// TIA Portal V18 export
FUNCTION_BLOCK "Utility_PID"   // FB2, FBD
TITLE = Utility PID Control
{ S7_Optimized_Access := 'TRUE' }
VERSION : 0.1
// Utility PID Control
// stored: AutoNumber true, IsIECCheckEnabled false, IsRetainMemResEnabled false, MemoryReserve 100, SetENOAutomatically false, UDAEnableTagReadback false
   VAR_INPUT
      START : Bool;
      SP : Real;
      PV : Real;
      CONTROL_MODE : Int;
      "TIME" : Int;
      PRE_SP : Int;
      AM : Bool;
      P : Int;
      I : Int;
      D : Int;
      JAC_IN : Real;
      JAC_OUT : Real;
      HHSP : Real;
      HSP : Real;
      LSP : Real;
      LLSP : Real;
      PIDRST : Bool;
      SOURCE_SEL : Int;
      AIR_XV_OPN : Bool;
      BYP_XV_OPN : Bool;
      VENT_OPN : Bool;
      CONDENSATE_XV_OPN : Bool;
      DRAIN_XV_OPN : Bool;
      SCV_XV_OPN : Bool;
   END_VAR
   VAR_OUTPUT
      START_PV : Real;
      CVOUT : Int;
      SCVOUT : Real;
      STATUS : Int;
      RAMP_SP : Real;
      JSP : Real;
      PID_PV : Real;
      RUN_MIN : Int;
      RUN_HR : Int;
      STEAM_SCVOUT : Real;
      STEAM_CVOUT : Int;
   END_VAR
   VAR_IN_OUT
      PAUSE : Bool;
      MAN_OUT : Real;
      TEMP_LIMIT : Real;
      STEAM_MAN_OUT : Real;
   END_VAR
   VAR
      RAMP_MODE : Bool;
      MAINT_MODE : Bool;
      J_MAINT_MODE : Bool;
      NO_RAMP : Bool;
      HEAT_COOL : Bool;
      BSTBIT : Bool;
      HOLD : Int;
      RAMP : Real;
      RAMP_RST : Bool;
      RMPSTART : Bool;
      Ramp_Substitute : Real;
      RAMP_INIT_RST : Bool;
      JKT_RAMP : Bool;
      MASS_CONTROL : Bool;
      TIMER_TRIG : Bool;
      iSTEAM_SCVOUT : Real;
      iSTEAM_CVOUT : Int;
      iSTEAM_SCV_SCL : Real;
      iSTEAM_CV_SCL : Int;
      iDRAIN_UP : Bool;
   END_VAR
BEGIN

REGION Network 1: Mode Selection
   // Mode Selection
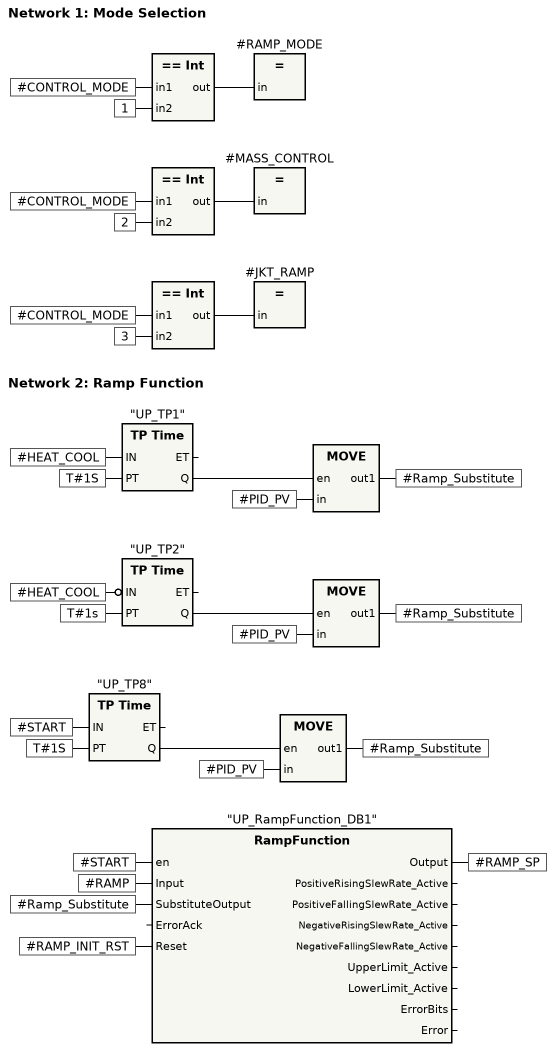
   #RAMP_MODE := #CONTROL_MODE = 1;
   #MASS_CONTROL := #CONTROL_MODE = 2;
   #JKT_RAMP := #CONTROL_MODE = 3;
END_REGION

REGION Network 2: Ramp Function
   // Ramp Function
   "UP_TP1".TP(IN := #HEAT_COOL, PT := T#1S);
   IF "UP_TP1".Q THEN #Ramp_Substitute := #PID_PV; END_IF;
   "UP_TP2".TP(IN := NOT #HEAT_COOL, PT := T#1s);
   IF "UP_TP2".Q THEN #Ramp_Substitute := #PID_PV; END_IF;
   "UP_TP8".TP(IN := #START, PT := T#1S);
   IF "UP_TP8".Q THEN #Ramp_Substitute := #PID_PV; END_IF;
   IF #START THEN
       "UP_RampFunction_DB1"(Input := #RAMP,   // RampFunction
                             SubstituteOutput := #Ramp_Substitute,
                             Reset := #RAMP_INIT_RST,
                             Output => #RAMP_SP);
   END_IF;
END_REGION

REGION Network 3: Ramp Reset
   // Ramp Reset
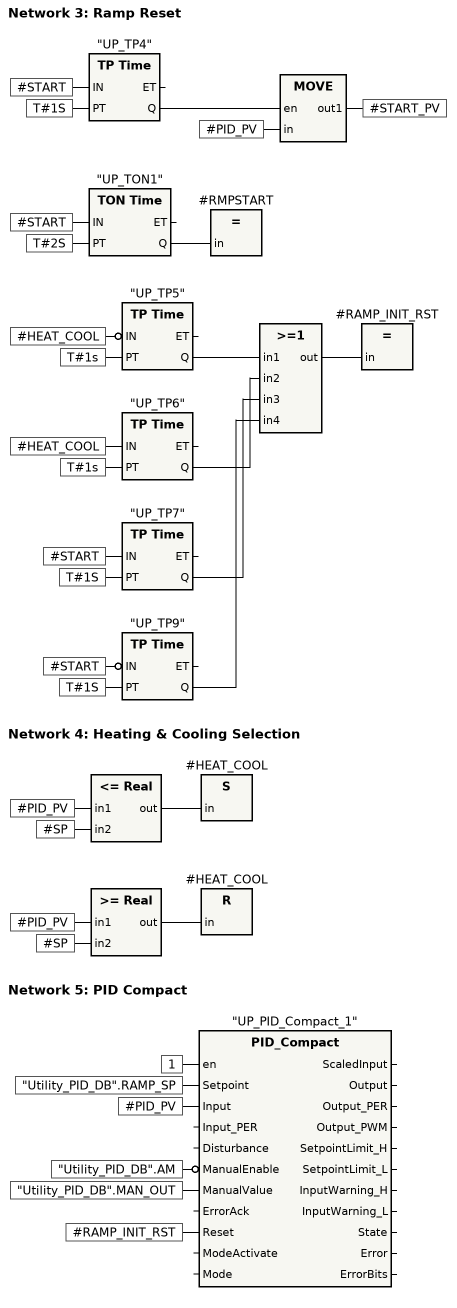
   "UP_TP4".TP(IN := #START, PT := T#1S);
   IF "UP_TP4".Q THEN #START_PV := #PID_PV; END_IF;
   "UP_TON1".TON(IN := #START, PT := T#2S);
   #RMPSTART := "UP_TON1".Q;
   "UP_TP5".TP(IN := NOT #HEAT_COOL, PT := T#1s);
   "UP_TP6".TP(IN := #HEAT_COOL, PT := T#1s);
   "UP_TP7".TP(IN := #START, PT := T#1S);
   "UP_TP9".TP(IN := NOT #START, PT := T#1S);
   #RAMP_INIT_RST := "UP_TP5".Q OR "UP_TP6".Q OR "UP_TP7".Q OR "UP_TP9".Q;
END_REGION

REGION Network 4: Heating & Cooling Selection
   // Heating & Cooling Selection
   IF #PID_PV <= #SP THEN #HEAT_COOL := TRUE; END_IF;
   IF #PID_PV >= #SP THEN #HEAT_COOL := FALSE; END_IF;
END_REGION

REGION Network 5: PID Compact
   IF 1 THEN
       "UP_PID_Compact_1"(Setpoint := "Utility_PID_DB".RAMP_SP,   // PID_Compact
                          Input := #PID_PV,
                          ManualEnable := NOT "Utility_PID_DB".AM,
                          ManualValue := "Utility_PID_DB".MAN_OUT,
                          Reset := #RAMP_INIT_RST);
   END_IF;
END_REGION

REGION Network 6 (SCL): Moving
   (* PID Parameters Moving *)
   "UP_PID_Compact_1".Retain.CtrlParams.Gain:= #P;
   "UP_PID_Compact_1".Retain.CtrlParams.Ti := #I;
   "UP_PID_Compact_1".Retain.CtrlParams.Td := #D;

   #RAMP := #SP;

   IF #RAMP_MODE OR #MASS_CONTROL THEN
       #PID_PV := #PV;
   END_IF;
   IF #JKT_RAMP THEN
       #PID_PV := #JAC_IN;
   END_IF;


   IF #AM = 1 AND #START = 1 AND #SOURCE_SEL<>5 THEN
       #SCVOUT := "UP_PID_Compact_1".Output;
       #CVOUT := "UP_PID_Compact_1".Output_PER;
   END_IF;
   IF (#AM = 1 AND #START = 0 ) OR (#AM = 1 AND #SOURCE_SEL=5) OR (#AM = 1 AND #START=1 AND (#AIR_XV_OPN OR #VENT_OPN OR #DRAIN_XV_OPN)) THEN
       #SCVOUT := 0.0;
       #CVOUT := 0;
   END_IF;
   IF #AM = 0 THEN
       #SCVOUT := "UP_PID_Compact_1".Output;
       #CVOUT := "UP_PID_Compact_1".Output_PER;
   END_IF;

   IF #AM = 1 AND #START = 1 AND #DRAIN_XV_OPN AND #SCV_XV_OPN THEN
       #iSTEAM_SCVOUT := 100.0;
       #iDRAIN_UP := 1;
   ELSE
       #iDRAIN_UP := 0;
   END_IF;
   IF #AM = 1 AND #START = 1 AND #SOURCE_SEL = 5 AND #iDRAIN_UP= 0 THEN
       #iSTEAM_SCVOUT := "UP_PID_Compact_1".Output;
       #iSTEAM_CVOUT := "UP_PID_Compact_1".Output_PER;
   END_IF;
   IF (#AM = 1 AND #START = 0) OR (#AM = 1 AND #SOURCE_SEL <> 5) OR (#AM = 1 AND #START = 1 AND ((#CONDENSATE_XV_OPN AND #SOURCE_SEL <> 5) OR (#AIR_XV_OPN AND #SOURCE_SEL = 5))) THEN
       #iSTEAM_SCVOUT := 0.0;
       #iSTEAM_CVOUT := 0;
   END_IF;


   (* Cooling *)
   IF #HEAT_COOL = 0 AND #START = 1 AND (#RAMP_MODE OR #JKT_RAMP) THEN
       "UP_RampFunction_DB1".PositiveFallingSlewRate := ABS((#START_PV - #SP) / (#TIME*60)); 
       "UP_PID_Compact_1".Config.InvertControl := 1;
   END_IF;
   IF #HEAT_COOL = 0 AND #START = 1 AND #MASS_CONTROL THEN
       "UP_RampFunction_DB1".PositiveFallingSlewRate := ABS((#START_PV - #SP) / (1 * 60));
       "UP_PID_Compact_1".Config.InvertControl := 1;
   END_IF;

   (* Heating *)
   IF #HEAT_COOL = 1 AND #START = 1 AND (#RAMP_MODE OR #JKT_RAMP) THEN
       "UP_RampFunction_DB1".PositiveRisingSlewRate := ABS((#SP - #START_PV) / (#TIME*60)); 
       "UP_PID_Compact_1".Config.InvertControl := 0;
   END_IF;
   IF #HEAT_COOL = 1 AND #START = 1 AND #MASS_CONTROL THEN
       "UP_RampFunction_DB1".PositiveRisingSlewRate := ABS((#SP - #START_PV) / (1 * 60));
       "UP_PID_Compact_1".Config.InvertControl := 0;
   END_IF;
END_REGION

REGION Network 7: OPERATION RUNTIME
   // OPERATION RUNTIME
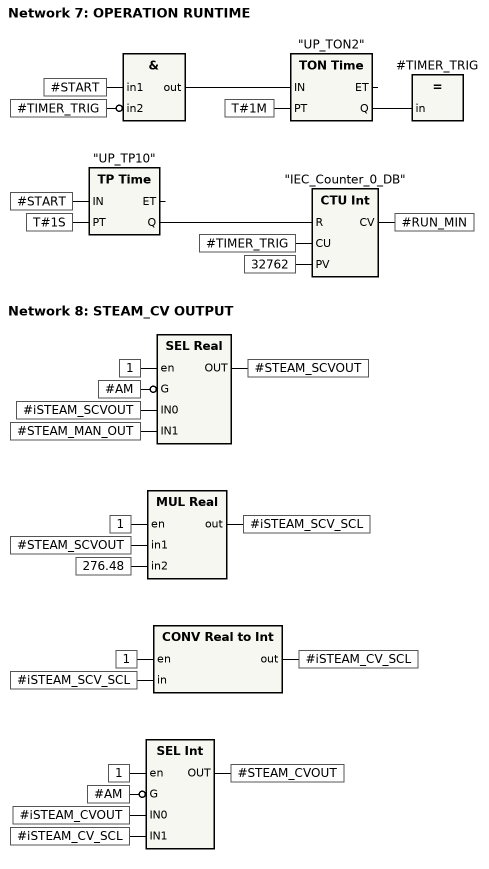
   "UP_TON2".TON(IN := #START AND NOT #TIMER_TRIG, PT := T#1M);
   #TIMER_TRIG := "UP_TON2".Q;
   "UP_TP10".TP(IN := #START, PT := T#1S);
   "IEC_Counter_0_DB".CTU(R := "UP_TP10".Q, CU := #TIMER_TRIG, PV := 32762, CV => #RUN_MIN);
END_REGION

REGION Network 8: STEAM_CV OUTPUT
   IF 1 THEN
       #STEAM_SCVOUT := SEL(G := NOT #AM, IN0 := #iSTEAM_SCVOUT, IN1 := #STEAM_MAN_OUT);
       #iSTEAM_SCV_SCL := #STEAM_SCVOUT * 276.48;
       #iSTEAM_CV_SCL := REAL_TO_INT(#iSTEAM_SCV_SCL);
       #STEAM_CVOUT := SEL(G := NOT #AM, IN0 := #iSTEAM_CVOUT, IN1 := #iSTEAM_CV_SCL);
   END_IF;
END_REGION
END_FUNCTION_BLOCK
